(* IEC 61131-3 sources: moenifar/, 2 files *)

(* ---- FB_LineSpeedControl.st ---- *)
(******************************************************************************
* فانکشن‌بلاک کنترل سرعت خط تولید / Line Speed Control Function Block
* ===========================================================================
* نام / Name: FB_LineSpeedControl
* نسخه / Version: 2.0 (بهینه‌سازی شده / Optimized)
* تاریخ / Date: 2025/01/07
*
* توضیحات / Description:
* این فانکشن‌بلاک برای کنترل دقیق سرعت خطوط تولید صنعتی طراحی شده است
* This function block is designed for precise control of industrial production line speeds
*
* کاربردها / Applications:
* - خطوط لمینیت / Laminate production lines
* - ماشین‌های چاپ / Printing machines
* - خطوط بسته‌بندی / Packaging lines
* - سیستم‌های نوار نقاله / Conveyor systems
* - خطوط نساجی / Textile production lines
*
* ویژگی‌های بهبود یافته / Enhanced Features:
* - حافظه سرعت قبل از توقف / Speed memory before stop
* - محاسبه شتاب لحظه‌ای / Instantaneous acceleration calculation
* - شمارنده زمان کارکرد / Runtime counter
* - هشدارهای سرعت / Speed warnings
* - محافظت از تغییرات ناگهانی / Sudden change protection
*******************************************************************************)

FUNCTION_BLOCK FB_LineSpeedControl

(* ===== ورودی‌ها / INPUTS ===== *)
VAR_INPUT
    (* کنترل اصلی / Main Control *)
    enable              : BOOL;             // فعال‌سازی فانکشن‌بلاک / Enable function block
    reset               : BOOL;             // ریست خطاها و قفل‌ها / Reset errors and latches

    (* انتخاب حالت / Mode Selection *)
    mode                : INT;              // حالت کار / Operating mode: 0=Manual, 1=HMI, 2=Auto

    (* نقاط تنظیم / Setpoints *)
    setpointHMI         : REAL;             // نقطه تنظیم از HMI / HMI setpoint (m/min)
    autoSetpoint        : REAL;             // نقطه تنظیم اتوماتیک / Automatic setpoint (m/min)

    (* کنترل دستی / Manual Control *)
    speedUp             : BOOL;             // دکمه افزایش سرعت / Speed up button
    speedDown           : BOOL;             // دکمه کاهش سرعت / Speed down button
    jogForward          : BOOL;             // حرکت آهسته رو به جلو / Jog forward
    jogReverse          : BOOL;             // حرکت آهسته رو به عقب / Jog reverse

    (* ایمنی / Safety *)
    stopEmergency       : BOOL;             // توقف اضطراری / Emergency stop
    safetyInterlockOK   : BOOL := TRUE;    // اینترلاک ایمنی / Safety interlock

    (* محدودیت‌ها / Limits *)
    maxSpeed            : REAL := 100.0;    // حداکثر سرعت مجاز / Maximum allowed speed (m/min)
    minSpeed            : REAL := 0.0;      // حداقل سرعت مجاز / Minimum allowed speed (m/min)
    jogSpeed            : REAL := 5.0;      // سرعت حرکت آهسته / Jog speed (m/min)

    (* پارامترهای رمپ / Ramp Parameters *)
    rampUpTimeNormal_s  : REAL := 5.0;     // زمان افزایش سرعت عادی / Normal ramp up time (s)
    rampDownTimeNormal_s: REAL := 5.0;     // زمان کاهش سرعت عادی / Normal ramp down time (s)
    rampDownTimeEmergency_s : REAL := 2.0; // زمان توقف اضطراری / Emergency stop time (s)
    manualRampTime_s    : REAL := 1.0;     // زمان رمپ دستی / Manual ramp time (s)
    rampStep            : REAL := 1.0;      // قدم تغییر سرعت دستی / Manual speed step (m/min)

    (* تنظیمات سیستم / System Settings *)
    scanCycle_ms        : REAL := 10.0;    // زمان چرخه اسکن PLC / PLC scan cycle time (ms)
    speedTolerance      : REAL := 0.5;      // تلرانس سرعت / Speed tolerance (m/min)
    warningThreshold    : REAL := 90.0;     // آستانه هشدار سرعت / Speed warning threshold (%)
END_VAR

(* ===== خروجی‌ها / OUTPUTS ===== *)
VAR_OUTPUT
    (* خروجی‌های اصلی / Main Outputs *)
    speedOut_mpm        : REAL;             // سرعت خروجی / Output speed (m/min)
    speedOut_percent    : REAL;             // سرعت خروجی درصدی / Output speed percentage (%)
    acceleration_mps2   : REAL;             // شتاب لحظه‌ای / Instantaneous acceleration (m/s²)

    (* وضعیت‌ها / Status *)
    isRunning           : BOOL;             // در حال کار / Running status
    atSetpoint          : BOOL;             // رسیدن به نقطه تنظیم / At setpoint
    emergencyLatched    : BOOL;             // قفل توقف اضطراری / Emergency stop latched

    (* هشدارها / Warnings *)
    speedWarning        : BOOL;             // هشدار سرعت بالا / High speed warning
    rampActive          : BOOL;             // رمپ فعال است / Ramp is active

    (* اطلاعات تشخیصی / Diagnostic Info *)
    currentMode         : STRING[20];       // نمایش حالت فعلی / Current mode display
    runTime_hours       : REAL;             // زمان کارکرد / Runtime hours
    totalDistance_km    : REAL;             // مسافت کل طی شده / Total distance traveled (km)
END_VAR

(* ===== متغیرهای داخلی / INTERNAL VARIABLES ===== *)
VAR
    (* متغیرهای کنترل / Control Variables *)
    targetSpeed         : REAL;             // سرعت هدف / Target speed
    previousSpeed       : REAL;             // سرعت قبلی / Previous speed
    speedBeforeStop     : REAL;             // سرعت قبل از توقف / Speed before stop
    manualSetpoint      : REAL;             // نقطه تنظیم دستی / Manual setpoint

    (* محاسبات رمپ / Ramp Calculations *)
    delta               : REAL;             // تفاوت سرعت / Speed difference
    step                : REAL;             // قدم رمپ / Ramp step
    rampTime            : REAL;             // زمان رمپ فعلی / Current ramp time
    actualRampRate      : REAL;             // نرخ واقعی رمپ / Actual ramp rate

    (* تایمرها و شمارنده‌ها / Timers & Counters *)
    runTimer            : TON;              // تایمر زمان کارکرد / Runtime timer
    distanceAccumulator : REAL;             // انباشتگر مسافت / Distance accumulator

    (* فلگ‌های کنترل / Control Flags *)
    firstScan           : BOOL := TRUE;     // اولین اسکن / First scan flag
    modeChanged         : BOOL;             // تغییر حالت / Mode changed flag
    previousMode        : INT;              // حالت قبلی / Previous mode
END_VAR

(* ===== کنستانت‌ها / CONSTANTS ===== *)
VAR CONSTANT
    MODE_MANUAL         : INT := 0;         // کد حالت دستی / Manual mode code
    MODE_HMI            : INT := 1;         // کد حالت HMI / HMI mode code
    MODE_AUTO           : INT := 2;         // کد حالت اتوماتیک / Auto mode code
    MIN_RAMP_TIME       : REAL := 0.1;      // حداقل زمان رمپ / Minimum ramp time (s)
    SPEED_ZERO_THRESHOLD: REAL := 0.1;      // آستانه سرعت صفر / Zero speed threshold
END_VAR

(* ========================================================================= *)
(* بدنه اصلی برنامه / MAIN PROGRAM BODY *)
(* ========================================================================= *)

(* ----- مقداردهی اولیه / Initialization ----- *)
IF firstScan THEN
    manualSetpoint := 0.0;
    speedOut_mpm := 0.0;
    previousSpeed := 0.0;
    runTime_hours := 0.0;
    totalDistance_km := 0.0;
    firstScan := FALSE;
END_IF;

(* ----- ریست خطاها / Reset Errors ----- *)
IF reset AND emergencyLatched THEN
    emergencyLatched := FALSE;
    speedBeforeStop := 0.0;
END_IF;

(* ----- بررسی فعال‌سازی و اینترلاک ایمنی / Check Enable & Safety Interlock ----- *)
IF NOT enable OR NOT safetyInterlockOK THEN
    (* کاهش تدریجی سرعت تا صفر / Gradual speed reduction to zero *)
    IF speedOut_mpm > SPEED_ZERO_THRESHOLD THEN
        speedOut_mpm := speedOut_mpm - SafeDivide(speedOut_mpm, rampDownTimeNormal_s * 1000.0 / scanCycle_ms);
    ELSE
        speedOut_mpm := 0.0;
    END_IF;
    isRunning := FALSE;
    currentMode := 'DISABLED';
    RETURN;
END_IF;

(* ----- مدیریت توقف اضطراری / Emergency Stop Management ----- *)
IF stopEmergency THEN
    (* ذخیره سرعت قبل از توقف / Save speed before stop *)
    IF NOT emergencyLatched AND speedOut_mpm > SPEED_ZERO_THRESHOLD THEN
        speedBeforeStop := speedOut_mpm;
    END_IF;

    (* کاهش سریع سرعت با رمپ اضطراری / Rapid speed reduction with emergency ramp *)
    speedOut_mpm := speedOut_mpm - SafeDivide(speedOut_mpm, rampDownTimeEmergency_s * 1000.0 / scanCycle_ms);

    (* قفل کردن سیستم پس از توقف کامل / Lock system after complete stop *)
    IF speedOut_mpm < SPEED_ZERO_THRESHOLD THEN
        speedOut_mpm := 0.0;
        emergencyLatched := TRUE;
        isRunning := FALSE;
    END_IF;

    currentMode := 'EMERGENCY STOP';
    RETURN;
END_IF;

(* ----- بررسی قفل اضطراری / Check Emergency Latch ----- *)
IF emergencyLatched THEN
    speedOut_mpm := 0.0;
    isRunning := FALSE;
    currentMode := 'E-STOP LATCHED';
    RETURN;
END_IF;

(* ----- مدیریت حرکت آهسته (Jog) / Jog Management ----- *)
IF jogForward OR jogReverse THEN
    IF jogForward AND NOT jogReverse THEN
        targetSpeed := jogSpeed;
        currentMode := 'JOG FORWARD';
    ELSIF jogReverse AND NOT jogForward THEN
        targetSpeed := -jogSpeed;
        currentMode := 'JOG REVERSE';
    ELSE
        (* هر دو دکمه فشرده شده - توقف / Both buttons pressed - stop *)
        targetSpeed := 0.0;
        currentMode := 'JOG CONFLICT';
    END_IF;
    rampTime := manualRampTime_s;

(* ----- انتخاب حالت عملکرد / Operating Mode Selection ----- *)
ELSE
    (* تشخیص تغییر حالت / Detect mode change *)
    IF mode <> previousMode THEN
        modeChanged := TRUE;
        previousMode := mode;
    ELSE
        modeChanged := FALSE;
    END_IF;

    (* تغییر خودکار به حالت دستی با فشردن دکمه‌ها / Auto switch to manual with button press *)
    IF (speedUp OR speedDown) AND (mode <> MODE_MANUAL) THEN
        mode := MODE_MANUAL;
        manualSetpoint := speedOut_mpm;
        modeChanged := TRUE;
    END_IF;

    (* پردازش حالت‌های مختلف / Process different modes *)
    CASE mode OF
        MODE_MANUAL:  (* حالت دستی / Manual Mode *)
            (* مدیریت دکمه‌های افزایش/کاهش سرعت / Handle speed up/down buttons *)
            IF speedUp AND NOT speedDown THEN
                manualSetpoint := manualSetpoint + rampStep;
            ELSIF speedDown AND NOT speedUp THEN
                manualSetpoint := manualSetpoint - rampStep;
            END_IF;

            (* اعمال محدودیت‌ها به setpoint دستی / Apply limits to manual setpoint *)
            manualSetpoint := LIMIT(minSpeed, manualSetpoint, maxSpeed);

            targetSpeed := manualSetpoint;
            rampTime := manualRampTime_s;
            currentMode := 'MANUAL';

        MODE_HMI:  (* حالت HMI / HMI Mode *)
            targetSpeed := LIMIT(minSpeed, setpointHMI, maxSpeed);
            rampTime := rampUpTimeNormal_s;
            currentMode := 'HMI CONTROL';

        MODE_AUTO:  (* حالت اتوماتیک / Auto Mode *)
            targetSpeed := LIMIT(minSpeed, autoSetpoint, maxSpeed);
            rampTime := rampUpTimeNormal_s;
            currentMode := 'AUTOMATIC';

        ELSE  (* حالت نامعتبر / Invalid mode *)
            targetSpeed := 0.0;
            currentMode := 'INVALID MODE';
    END_CASE;
END_IF;

(* ----- محاسبه و اعمال رمپ سرعت / Calculate and Apply Speed Ramp ----- *)
(* محاسبه اختلاف سرعت / Calculate speed difference *)
delta := targetSpeed - speedOut_mpm;

(* انتخاب زمان رمپ بر اساس جهت تغییر / Select ramp time based on direction *)
IF delta > 0 THEN
    (* افزایش سرعت / Speed increase *)
    rampTime := MAX(MIN_RAMP_TIME, rampUpTimeNormal_s);
ELSIF delta < 0 THEN
    (* کاهش سرعت / Speed decrease *)
    rampTime := MAX(MIN_RAMP_TIME, rampDownTimeNormal_s);
END_IF;

(* محاسبه قدم رمپ / Calculate ramp step *)
IF ABS(delta) > speedTolerance THEN
    step := SafeDivide(delta, rampTime * 1000.0 / scanCycle_ms);
    speedOut_mpm := speedOut_mpm + step;
    rampActive := TRUE;
ELSE
    (* رسیدن به نقطه تنظیم / Reached setpoint *)
    speedOut_mpm := targetSpeed;
    rampActive := FALSE;
END_IF;

(* ----- اعمال محدودیت‌های نهایی / Apply Final Limits ----- *)
speedOut_mpm := LIMIT(minSpeed, speedOut_mpm, maxSpeed);

(* ----- محاسبات خروجی / Output Calculations ----- *)
(* محاسبه درصد سرعت / Calculate speed percentage *)
IF maxSpeed > 0 THEN
    speedOut_percent := (speedOut_mpm / maxSpeed) * 100.0;
ELSE
    speedOut_percent := 0.0;
END_IF;

(* محاسبه شتاب / Calculate acceleration *)
(* شتاب = تغییر سرعت / زمان *)
(* Acceleration = speed change / time *)
IF scanCycle_ms > 0 THEN
    acceleration_mps2 := ((speedOut_mpm - previousSpeed) / 60.0) / (scanCycle_ms / 1000.0);
ELSE
    acceleration_mps2 := 0.0;
END_IF;

(* به‌روزرسانی سرعت قبلی / Update previous speed *)
previousSpeed := speedOut_mpm;

(* ----- تنظیم وضعیت‌ها / Set Status Flags ----- *)
(* وضعیت در حال کار / Running status *)
isRunning := ABS(speedOut_mpm) > SPEED_ZERO_THRESHOLD;

(* رسیدن به نقطه تنظیم / At setpoint *)
atSetpoint := ABS(speedOut_mpm - targetSpeed) <= speedTolerance;

(* هشدار سرعت بالا / High speed warning *)
speedWarning := speedOut_percent >= warningThreshold;

(* ----- محاسبات زمان کارکرد و مسافت / Runtime and Distance Calculations ----- *)
(* تایمر زمان کارکرد / Runtime timer *)
runTimer(IN := isRunning, PT := T#1H);
IF runTimer.Q THEN
    runTime_hours := runTime_hours + 1.0;
    runTimer(IN := FALSE);  (* ریست تایمر / Reset timer *)
END_IF;

(* محاسبه مسافت طی شده / Calculate distance traveled *)
(* مسافت = سرعت × زمان *)
(* Distance = speed × time *)
IF isRunning THEN
    distanceAccumulator := distanceAccumulator + (ABS(speedOut_mpm) * scanCycle_ms / 60000.0);
    IF distanceAccumulator >= 1000.0 THEN
        totalDistance_km := totalDistance_km + 1.0;
        distanceAccumulator := distanceAccumulator - 1000.0;
    END_IF;
END_IF;

END_FUNCTION_BLOCK

(******************************************************************************
* تابع تقسیم ایمن / Safe Division Function
* ===========================================================================
* این تابع از خطای تقسیم بر صفر جلوگیری می‌کند
* This function prevents division by zero errors
*******************************************************************************)
FUNCTION SafeDivide : REAL
VAR_INPUT
    numerator   : REAL;     // صورت کسر / Numerator
    denominator : REAL;     // مخرج کسر / Denominator
END_VAR

VAR
    ZERO_THRESHOLD : REAL := 0.0001;  // آستانه صفر / Zero threshold
END_VAR

(* بررسی مخرج برای جلوگیری از تقسیم بر صفر / Check denominator to prevent division by zero *)
IF ABS(denominator) < ZERO_THRESHOLD THEN
    (* بازگشت صفر در صورت مخرج صفر / Return zero if denominator is zero *)
    SafeDivide := 0.0;
ELSE
    (* انجام تقسیم عادی / Perform normal division *)
    SafeDivide := numerator / denominator;
END_IF;

END_FUNCTION

(* ---- Example_Usage.st ---- *)
(******************************************************************************
* نمونه استفاده از فانکشن‌بلاک کنترل سرعت خط / Line Speed Control Usage Example
* ===========================================================================
* این برنامه نحوه استفاده از FB_LineSpeedControl را نشان می‌دهد
* This program demonstrates how to use FB_LineSpeedControl
*
* سناریوهای پوشش داده شده / Covered Scenarios:
* 1. کنترل دستی با دکمه‌ها / Manual control with buttons
* 2. کنترل از HMI / HMI control
* 3. کنترل اتوماتیک / Automatic control
* 4. توقف اضطراری و ریست / Emergency stop and reset
* 5. حرکت آهسته (Jog) / Jog operation
* 6. نمایش اطلاعات تشخیصی / Display diagnostic information
*******************************************************************************)

PROGRAM Example_LineSpeedControl

(* ===== متغیرهای ورودی از سیستم / Input Variables from System ===== *)
VAR
    (* دکمه‌های کنترل / Control Buttons *)
    btnEnable           : BOOL;             // دکمه فعال‌سازی / Enable button
    btnReset            : BOOL;             // دکمه ریست / Reset button
    btnEmergencyStop    : BOOL;             // دکمه توقف اضطراری / Emergency stop button
    btnSpeedUp          : BOOL;             // دکمه افزایش سرعت / Speed up button
    btnSpeedDown        : BOOL;             // دکمه کاهش سرعت / Speed down button
    btnJogForward       : BOOL;             // دکمه حرکت آهسته جلو / Jog forward button
    btnJogReverse       : BOOL;             // دکمه حرکت آهسته عقب / Jog reverse button

    (* انتخابگر حالت / Mode Selector *)
    modeSelector        : INT := 1;         // 0=Manual, 1=HMI, 2=Auto

    (* ورودی‌های HMI / HMI Inputs *)
    hmiSpeedSetpoint    : REAL := 50.0;    // نقطه تنظیم سرعت از HMI / Speed setpoint from HMI (m/min)

    (* ورودی‌های اتوماتیک / Automatic Inputs *)
    autoSpeedCommand    : REAL := 75.0;    // فرمان سرعت از سیستم بالادست / Speed command from higher system (m/min)

    (* سنسورها و فیدبک / Sensors & Feedback *)
    safetyGatesClosed   : BOOL := TRUE;    // وضعیت درب‌های ایمنی / Safety gates status
    motorTempOK         : BOOL := TRUE;    // دمای موتور نرمال / Motor temperature OK

    (* پارامترهای خط تولید / Production Line Parameters *)
    productType         : INT := 1;         // نوع محصول / Product type (1-5)
    lineLength          : REAL := 100.0;    // طول خط تولید / Production line length (m)
END_VAR

(* ===== پارامترهای قابل تنظیم / Configurable Parameters ===== *)
VAR
    (* تنظیمات برای انواع محصول / Settings for Product Types *)
    maxLineSpeed        : REAL := 120.0;    // حداکثر سرعت خط / Maximum line speed (m/min)
    minLineSpeed        : REAL := 5.0;      // حداقل سرعت خط / Minimum line speed (m/min)
    jogSpeedSetting     : REAL := 3.0;      // سرعت حرکت آهسته / Jog speed (m/min)

    (* زمان‌های رمپ / Ramp Times *)
    normalRampUp        : REAL := 10.0;     // زمان رمپ بالا عادی / Normal ramp up time (s)
    normalRampDown      : REAL := 8.0;      // زمان رمپ پایین عادی / Normal ramp down time (s)
    emergencyRampTime   : REAL := 3.0;      // زمان رمپ اضطراری / Emergency ramp time (s)
    manualRampTime      : REAL := 0.5;      // زمان رمپ دستی / Manual ramp time (s)

    (* تنظیمات سیستم / System Settings *)
    plcScanTime         : REAL := 20.0;     // زمان اسکن PLC / PLC scan time (ms)
    speedStep           : REAL := 2.0;      // قدم تغییر سرعت دستی / Manual speed step (m/min)
    speedToleranceBand  : REAL := 1.0;      // باند تلرانس سرعت / Speed tolerance band (m/min)
    highSpeedWarning    : REAL := 85.0;     // آستانه هشدار سرعت بالا / High speed warning threshold (%)
END_VAR

(* ===== اینستنس فانکشن‌بلاک / Function Block Instance ===== *)
VAR
    lineSpeedController : FB_LineSpeedControl;  // کنترلر سرعت خط / Line speed controller
END_VAR

(* ===== متغیرهای خروجی برای نمایش / Output Variables for Display ===== *)
VAR
    (* اطلاعات سرعت / Speed Information *)
    actualSpeed         : REAL;             // سرعت واقعی / Actual speed (m/min)
    speedPercentage     : REAL;             // سرعت به درصد / Speed percentage (%)
    currentAcceleration : REAL;             // شتاب فعلی / Current acceleration (m/s²)

    (* وضعیت‌ها / Status *)
    lineRunning         : BOOL;             // خط در حال کار / Line running
    speedReached        : BOOL;             // رسیدن به سرعت هدف / Target speed reached
    emergencyActive     : BOOL;             // توقف اضطراری فعال / Emergency stop active
    rampInProgress      : BOOL;             // رمپ در حال اجرا / Ramp in progress
    highSpeedAlarm      : BOOL;             // آلارم سرعت بالا / High speed alarm

    (* اطلاعات عملیاتی / Operational Information *)
    operatingMode       : STRING[20];       // حالت عملیاتی / Operating mode
    totalRunTime        : REAL;             // زمان کل کارکرد / Total runtime (hours)
    totalDistance       : REAL;             // مسافت کل / Total distance (km)

    (* محاسبات کارایی / Efficiency Calculations *)
    averageSpeed        : REAL;             // سرعت متوسط / Average speed (m/min)
    productionRate      : REAL;             // نرخ تولید / Production rate (units/hour)
END_VAR

(* ===== منطق برای تعیین اینترلاک ایمنی / Safety Interlock Logic ===== *)
VAR
    safetyInterlock     : BOOL;             // اینترلاک ایمنی کلی / Overall safety interlock
END_VAR

(* ========================================================================= *)
(* بدنه اصلی برنامه / MAIN PROGRAM BODY *)
(* ========================================================================= *)

(* ----- تنظیم پارامترها بر اساس نوع محصول / Set Parameters Based on Product Type ----- *)
CASE productType OF
    1:  (* محصول نوع 1 - سرعت پایین / Product Type 1 - Low Speed *)
        maxLineSpeed := 60.0;
        normalRampUp := 5.0;
        normalRampDown := 4.0;

    2:  (* محصول نوع 2 - سرعت متوسط / Product Type 2 - Medium Speed *)
        maxLineSpeed := 100.0;
        normalRampUp := 8.0;
        normalRampDown := 6.0;

    3:  (* محصول نوع 3 - سرعت بالا / Product Type 3 - High Speed *)
        maxLineSpeed := 150.0;
        normalRampUp := 12.0;
        normalRampDown := 10.0;

    4:  (* محصول نوع 4 - محصول حساس / Product Type 4 - Sensitive Product *)
        maxLineSpeed := 80.0;
        normalRampUp := 15.0;
        normalRampDown := 12.0;
        emergencyRampTime := 5.0;

    5:  (* محصول نوع 5 - تولید سریع / Product Type 5 - Fast Production *)
        maxLineSpeed := 200.0;
        normalRampUp := 10.0;
        normalRampDown := 8.0;
        speedStep := 5.0;

    ELSE  (* پیش‌فرض / Default *)
        maxLineSpeed := 100.0;
        normalRampUp := 10.0;
        normalRampDown := 8.0;
END_CASE;

(* ----- محاسبه اینترلاک ایمنی / Calculate Safety Interlock ----- *)
safetyInterlock := safetyGatesClosed AND motorTempOK;

(* ----- فراخوانی فانکشن‌بلاک کنترل سرعت / Call Line Speed Control Function Block ----- *)
lineSpeedController(
    (* ورودی‌های کنترل اصلی / Main Control Inputs *)
    enable              := btnEnable,
    reset               := btnReset,
    mode                := modeSelector,

    (* نقاط تنظیم / Setpoints *)
    setpointHMI         := hmiSpeedSetpoint,
    autoSetpoint        := autoSpeedCommand,

    (* کنترل دستی / Manual Control *)
    speedUp             := btnSpeedUp,
    speedDown           := btnSpeedDown,
    jogForward          := btnJogForward,
    jogReverse          := btnJogReverse,

    (* ایمنی / Safety *)
    stopEmergency       := btnEmergencyStop,
    safetyInterlockOK   := safetyInterlock,

    (* محدودیت‌ها / Limits *)
    maxSpeed            := maxLineSpeed,
    minSpeed            := minLineSpeed,
    jogSpeed            := jogSpeedSetting,

    (* پارامترهای رمپ / Ramp Parameters *)
    rampUpTimeNormal_s  := normalRampUp,
    rampDownTimeNormal_s:= normalRampDown,
    rampDownTimeEmergency_s := emergencyRampTime,
    manualRampTime_s    := manualRampTime,
    rampStep            := speedStep,

    (* تنظیمات سیستم / System Settings *)
    scanCycle_ms        := plcScanTime,
    speedTolerance      := speedToleranceBand,
    warningThreshold    := highSpeedWarning
);

(* ----- خواندن خروجی‌ها / Read Outputs ----- *)
(* اطلاعات سرعت / Speed Information *)
actualSpeed         := lineSpeedController.speedOut_mpm;
speedPercentage     := lineSpeedController.speedOut_percent;
currentAcceleration := lineSpeedController.acceleration_mps2;

(* وضعیت‌ها / Status *)
lineRunning         := lineSpeedController.isRunning;
speedReached        := lineSpeedController.atSetpoint;
emergencyActive     := lineSpeedController.emergencyLatched;
rampInProgress      := lineSpeedController.rampActive;
highSpeedAlarm      := lineSpeedController.speedWarning;

(* اطلاعات عملیاتی / Operational Information *)
operatingMode       := lineSpeedController.currentMode;
totalRunTime        := lineSpeedController.runTime_hours;
totalDistance       := lineSpeedController.totalDistance_km;

(* ----- محاسبات اضافی / Additional Calculations ----- *)
(* محاسبه سرعت متوسط / Calculate Average Speed *)
IF totalRunTime > 0 THEN
    averageSpeed := (totalDistance * 1000.0) / (totalRunTime * 60.0);  // m/min
ELSE
    averageSpeed := 0.0;
END_IF;

(* محاسبه نرخ تولید تخمینی / Calculate Estimated Production Rate *)
(* فرض: هر 10 متر خط = 1 واحد محصول / Assumption: Every 10m of line = 1 product unit *)
IF lineRunning AND actualSpeed > 0 THEN
    productionRate := (actualSpeed * 60.0) / 10.0;  // units/hour
ELSE
    productionRate := 0.0;
END_IF;

(* ----- نمایش اطلاعات تشخیصی در HMI / Display Diagnostic Info on HMI ----- *)
(* این اطلاعات می‌تواند در HMI نمایش داده شود *)
(* This information can be displayed on HMI *)

(*
مثال نمایش در HMI / HMI Display Example:
=====================================
سرعت فعلی / Current Speed: [actualSpeed] m/min ([speedPercentage]%)
شتاب / Acceleration: [currentAcceleration] m/s²
حالت عملیاتی / Operating Mode: [operatingMode]
وضعیت خط / Line Status: [IF lineRunning THEN "در حال کار/Running" ELSE "متوقف/Stopped"]
زمان کارکرد / Runtime: [totalRunTime] hours
مسافت طی شده / Distance: [totalDistance] km
سرعت متوسط / Avg Speed: [averageSpeed] m/min
نرخ تولید / Production Rate: [productionRate] units/hr

هشدارها / Warnings:
- سرعت بالا / High Speed: [highSpeedAlarm]
- توقف اضطراری / E-Stop: [emergencyActive]
- رمپ فعال / Ramp Active: [rampInProgress]
*)

END_PROGRAM
